Staubli VAL3: init.pgx

public program init(num& x_nError[])
  local bool l_bOk
  local num l_i
  local num l_j
  local num l_nCol
  local num l_nRow
  local num l_nValue
  local string l_sData[2]
begin
  //This program performs some checkings on the different variables
  // used for the Popupwindow definitions
  //
  // Input Param
  // None
  //
  // Output Param
  //  x_nError    : Error code
  //
  //Created 21/12/05                              C.CURRIVAND
  //--------------------------------------------------------------
  //
  // Check data integrity
  resize(nListSize,1,size(sTxtBoxCaption))
  for l_i=0 to size(sTxtBoxCaption)-1
    l_j=0
    // Check that sTxtBoxLen is numerical
    while (l_j<len(sTxtBoxLen[l_i])) and ((asc(sTxtBoxLen[l_i],l_j)>=48) and (asc(sTxtBoxLen[l_i],l_j)<=57))
      l_j=l_j+1
    endWhile
    //
    if l_j==len(sTxtBoxLen)
      // get textboxes position
      call ut:_str2Array(sTxtBoxPos[l_i],";",l_sData)
      toNum(l_sData[0],l_nCol,l_bOk)
      toNum(l_sData[1],l_nRow,l_bOk)
      // Check that textbox position is within the screen dimensions
      x_nError=0
      toNum(sTxtBoxLen[l_i],l_nValue[0],l_bOk)
      l_nCol=l_nCol+l_nValue
      if (l_nCol<0 or l_nCol>nCOLMAX) or (l_nRow<0 or l_nRow>nROWMAX)
        x_nError=-3
        call ut:addNumToString(sErrorMsg[-x_nError],sErrorMessage,"*",l_nValue)
        l_i=size(sTxtBoxCaption)
      endIf
    else
      x_nError=-2
      call ut:addNumToString(sErrorMsg[-x_nError],sErrorMessage,"*",l_i)
      l_i=size(sTxtBoxCaption)
    endIf
  endFor
end
